// TIA Portal project "WASH TON_TOM" (V19)

(* hardware
DEVICE "SIMATIC 1200 station_1"  S71200.Device
   slot 0: "S7-1200 rack"  Rack  V1.0
   slot 1: "PLC_1"  CPU 1214C DC/DC/DC  6ES7 214-1AG40-0XB0  V4.0
   slot 3: "AQ1 x 12 bits_1"  6ES7 232-4HA30-0XB0  V1.0
*)

// ===== PLC "PLC_1"  CPU 1214C DC/DC/DC =====

VAR_GLOBAL   // PLC tag table "Default tag table"
   "PUSHBUTTON" AT %I0.0 : Bool;   // Pushbutton Wash Cycle
   "SWITCH_CLAMP1" AT %I0.1 : Bool;   // Limit Switch Clamp 1
   "SWITCH_CLAMP2" AT %I0.2 : Bool;   // Limit Switch Clamp 2
   "SOLENOID_CLAMP1" AT %Q0.0 : Bool;   // Clamp 1 Solenoid
   "SOLENOID_CLAMP2" AT %Q0.1 : Bool;   // Clamp 2 Solenoid
   "WASH_VALVE" AT %Q0.2 : Bool;   // Spray Wash Valve
END_VAR

// folder: System blocks/Program resources

DATA_BLOCK "WASH_DELAY"   // DB1
{ S7_Optimized_Access := 'TRUE' }
AUTHOR : Simatic
FAMILY : IEC
NAME : IEC_TMR
VERSION : 1.0
// stored: InstanceOfName IEC_TIMER
"IEC_TIMER"
BEGIN
END_DATA_BLOCK

// folder: (top level)

ORGANIZATION_BLOCK "Main"   // OB1, FBD, ProgramCycle
TITLE = "Main Program Sweep (Cycle)"
{ S7_Optimized_Access := 'TRUE' }
VERSION : 0.1
BEGIN

REGION Network 1: Clamp 1 Solenoid
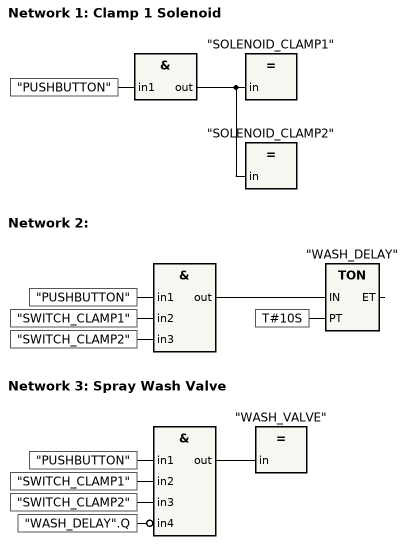
   "SOLENOID_CLAMP1" := "PUSHBUTTON";
   "SOLENOID_CLAMP2" := "PUSHBUTTON";
END_REGION

REGION Network 2
   "WASH_DELAY".TON(IN := "PUSHBUTTON" AND "SWITCH_CLAMP1" AND "SWITCH_CLAMP2", PT := T#10S);
END_REGION

REGION Network 3: Spray Wash Valve
   "WASH_VALVE" := "PUSHBUTTON" AND "SWITCH_CLAMP1" AND "SWITCH_CLAMP2" AND NOT "WASH_DELAY".Q;
END_REGION
END_ORGANIZATION_BLOCK